// TIA Portal project "NodeRed_0" (V20)

(* hardware
DEVICE "S7-1500/ET200MP-Station_1"  S7-1500 station
   slot 0: "Profilschiene_0"  Rack  6ES7 590-1***0-0AA0
   slot 1: "PLC_1"  CPU 1515-2 PN  6ES7 515-2AM02-0AB0  V2.9
      slot 3: "CPU-Display_1"  6ES7591-1BA00-0AA0
      slot 32768: "PROFINET-Schnittstelle_1"  X1
         slot 32769: "Port_1"  X1 P1
         slot 32770: "Port_2"  X1 P2
      slot 33024: "PROFINET-Schnittstelle_2"  X2
         slot 33025: "Port_1"  X2 P1
      slot 34817: "Virtual CP interface port_1"  Virtual CP interface port  Virtual CP interface port
DEVICE "HMI_1"  TP700 Comfort
   slot 0: "HMI_1"  TP700 Comfort  6AV2 124-0GC01-0AX0  17.0.0.0
   slot 1: "HMI_RT_1"  TP700 Comfort  6AV2 124-0GC01-0AX0  17.0.0.0
   slot 5: "HMI_1.IE_CP_1"  PROFINET Interface  17.0.0.0
      slot 1: "PROFINET Schnittstelle_1"  PROFINET Interface
         slot 1: "Port_1"  Port
         slot 2: "Port_2"  Port
   slot 7: "HMI_1.MPI/DP_CP_1"  MPI/DP Interface  17.0.0.0
*)

// ===== PLC "PLC_1"  CPU 1515-2 PN =====

VAR_GLOBAL   // PLC tag table "Eingaenge"
   "2B1" AT %ED30 : DInt;   // Visionsensor
   "1B1" AT %E0.0 : Bool;   // Sensor_ein
   "3B1" AT %E0.1 : Bool;   // Sensor_aus
   "Factory/IO Running" AT %E0.7 : Bool;
END_VAR

VAR_GLOBAL   // PLC tag table "Ausgaenge"
   "1M1" AT %A0.0 : Bool;   // Band_1 (2m)
   "2M1" AT %A0.1 : Bool;   // Band_2 (2m)
   "3M1" AT %A0.2 : Bool;   // Band_3 (2m)
   "D1" AT %AD30 : DInt;   // Display
   "1H1" AT %A0.6 : Bool;   // Meldeleuchte (rot)
   "1H3" AT %A0.7 : Bool;   // Meldeleuchte (grün)
END_VAR

TYPE "typEingaenge"
   STRUCT
      "1B1" : Bool;
      "2B1" : DInt;
      "3B1" : Bool;
   END_STRUCT;
END_TYPE

TYPE "typAusgaenge"
   STRUCT
      "1M1" : Bool;
      "2M1" : Bool;
      "3M1" : Bool;
   END_STRUCT;
END_TYPE

TYPE "typZaehler"
   STRUCT
      Gesamt : DInt;
      Blau : Struct
         Gesamt : DInt;
         Roh : DInt;
         Oberteil : DInt;
         Unterteil : DInt;
      END_STRUCT;
      Gruen : Struct
         Gesamt : DInt;
         Roh : DInt;
         Oberteil : DInt;
         Unterteil : DInt;
      END_STRUCT;
      Metall : Struct
         Gesamt : DInt;
         Roh : DInt;
         Oberteil : DInt;
         Unterteil : DInt;
      END_STRUCT;
   END_STRUCT;
END_TYPE

DATA_BLOCK "IDB_Anlage_ein"   // DB1
{ S7_Optimized_Access := 'TRUE' }
VERSION : 0.1
// stored: InstanceOfName Anlage_ein
"Anlage_ein"
BEGIN
END_DATA_BLOCK

DATA_BLOCK "IDB_Bandsteuerung"   // DB10
{ S7_Optimized_Access := 'TRUE' }
VERSION : 0.1
// stored: InstanceOfName Bandsteuerung
"Bandsteuerung"
BEGIN
END_DATA_BLOCK

DATA_BLOCK "IDB_Bauteile_zaehlen"   // DB20
{ S7_Optimized_Access := 'TRUE' }
VERSION : 0.1
// stored: InstanceOfName Bauteile_zaehlen
"Bauteile_zaehlen"
BEGIN
END_DATA_BLOCK

DATA_BLOCK "HMI"   // DB100
{ S7_Optimized_Access := 'TRUE' }
VERSION : 0.1
   VAR
      Eingaenge : "typEingaenge";
      Ausgaenge : "typAusgaenge";
      Anlagedaten : Struct
         Anlage_aktiv : Bool;
         Laufzeit : DTL;
         Bauteile : "typZaehler";
         Bauteil : DInt;
      END_STRUCT;
   END_VAR
BEGIN
END_DATA_BLOCK

FUNCTION_BLOCK "Anlage_ein"   // FB1, FBD
{ S7_Optimized_Access := 'TRUE' }
VERSION : 0.1
BEGIN

REGION Network 1 (SCL)
   "HMI".Eingaenge."1B1" := "1B1";
   "HMI".Eingaenge."2B1" := "2B1";
   "HMI".Eingaenge."3B1" := "3B1";
END_REGION
END_FUNCTION_BLOCK

FUNCTION_BLOCK "Bandsteuerung"   // FB10, FBD
{ S7_Optimized_Access := 'TRUE' }
VERSION : 0.1
   VAR
      MI_RTRIG_FactoryRun : R_TRIG;
      MI_FTRIG_1B1 : F_TRIG;
      MI_FTRIG_3B1 : F_TRIG;
   END_VAR
BEGIN

REGION Network 1 (SCL): Flanken
   #MI_RTRIG_FactoryRun(CLK:="Factory/IO Running");

   #MI_FTRIG_1B1(CLK:="HMI".Eingaenge."1B1");
   #MI_FTRIG_3B1(CLK := "HMI".Eingaenge."3B1");
END_REGION

REGION Network 2 (SCL)
   "HMI".Ausgaenge."1M1" :=
   "HMI".Ausgaenge."2M1" :=
   "HMI".Ausgaenge."3M1" := #MI_RTRIG_FactoryRun.Q;
END_REGION
END_FUNCTION_BLOCK

FUNCTION_BLOCK "Bauteile_zaehlen"   // FB20, FBD
{ S7_Optimized_Access := 'TRUE' }
VERSION : 0.1
   VAR_INPUT
      Trigger : Bool;
      Bauteil : DInt;
   END_VAR
   VAR_IN_OUT
      Anzahl : "typZaehler";
   END_VAR
BEGIN

REGION Network 1 (SCL)
   IF #Trigger THEN
       CASE #Bauteil OF
           // Blaue Teile
           1:
               #Anzahl.Blau.Roh += 1;
           2:
               #Anzahl.Blau.Oberteil += 1;
           3:
               #Anzahl.Blau.Unterteil += 1;

           // Grüne Teile
           4:
               #Anzahl.Gruen.Roh += 1;
           5:
               #Anzahl.Gruen.Oberteil += 1;
           6:
               #Anzahl.Gruen.Unterteil += 1;

           // Metall Teile
           4:
               #Anzahl.Metall.Roh += 1;
           5:
               #Anzahl.Metall.Oberteil += 1;
           6:
               #Anzahl.Metall.Unterteil += 1;
       END_CASE;


       // Gesamtnanzahl einzelne Teile
       #Anzahl.Blau.Gesamt := #Anzahl.Blau.Roh
                           + #Anzahl.Blau.Oberteil
                           + #Anzahl.Blau.Unterteil;

       #Anzahl.Gruen.Gesamt := #Anzahl.Gruen.Roh
                           + #Anzahl.Gruen.Oberteil
                           + #Anzahl.Gruen.Unterteil;

       #Anzahl.Metall.Gesamt := #Anzahl.Metall.Roh
                           + #Anzahl.Metall.Oberteil
                           + #Anzahl.Metall.Unterteil;


       // Gesamtnanzahl alle Teile
       #Anzahl.Gesamt := #Anzahl.Metall.Gesamt
                       + #Anzahl.Gruen.Gesamt
                       + #Anzahl.Metall.Gesamt;
   END_IF;
END_REGION
END_FUNCTION_BLOCK

FUNCTION "Anlage_aus" : Void   // FC1, FBD
{ S7_Optimized_Access := 'TRUE' }
VERSION : 0.1
BEGIN

REGION Network 1 (SCL)
   // Bits
   "1M1" := "HMI".Ausgaenge."1M1";
   "2M1" := "HMI".Ausgaenge."2M1";
   "3M1" := "HMI".Ausgaenge."3M1";

   "Tag_1" := NOT "HMI".Anlagedaten.Anlage_aktiv;
   "Tag_2" := "HMI".Anlagedaten.Anlage_aktiv;


   // Word
   "D1" := "HMI".Anlagedaten.Anzahl_Bauteile.Gesamt;
END_REGION
END_FUNCTION

ORGANIZATION_BLOCK "Main"   // OB1, FBD, ProgramCycle
TITLE = "Main Program Sweep (Cycle)"
{ S7_Optimized_Access := 'TRUE' }
VERSION : 0.1
   VAR_INPUT
      Initial_Call : Bool;   // Initial call of this OB
      Remanence : Bool;   // =True, if remanent data are available
   END_VAR
BEGIN

REGION Network 1
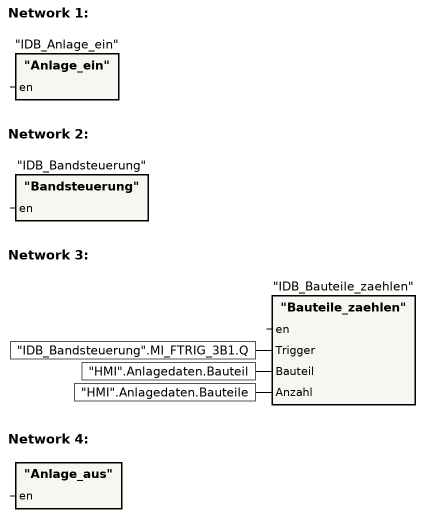
   "IDB_Anlage_ein"();   // "Anlage_ein"
END_REGION

REGION Network 2
   "IDB_Bandsteuerung"();   // "Bandsteuerung"
END_REGION

REGION Network 3
   "IDB_Bauteile_zaehlen"(Trigger := "IDB_Bandsteuerung".MI_FTRIG_3B1.Q,   // "Bauteile_zaehlen"
                          Bauteil := "HMI".Anlagedaten.Bauteil,
                          Anzahl := "HMI".Anlagedaten.Bauteile);
END_REGION

REGION Network 4
   "Anlage_aus"();
END_REGION
END_ORGANIZATION_BLOCK

(* ===== HMI "HMI_RT_1" =====
system functions are stored by id; their names below are inferred from use

HMI tags "Standard-Variablentabelle"
   "Variable_Bildnummer" : UInt, internal

text list "Textliste_Bildnamen": 1 'Home'; 2 'Anlagedaten'

screen "01_Home" 800x420, template "Menueleiste"
   on GenerateScreen: SetTag("Variable_Bildnummer", 1)

Template "Menueleiste" 800x420
   Button "Beenden" at 720,360 size 78x58; TextOff 'Beenden'; PictureOff "ExitRuntime_TP700_Comfort_TR"; PictureOn "ExitRuntime_TP700_Comfort_TR"
      on Release: StopRuntime(0)
   Button "Template_Button" at 640,360 size 78x58; TextOff 'Text'
   Button "Template_Button_1" at 560,360 size 78x58; TextOff 'Text'
   Button "Template_Button_2" at 480,360 size 78x58; TextOff 'Text'
   Button "Template_Button_3" at 400,360 size 78x58; TextOff 'Text'
   Button "Template_Button_4" at 321,360 size 78x58; TextOff 'Text'
   Button "Template_Button_5" at 241,360 size 78x58; TextOff 'Text'
   Button "Template_Button_6" at 161,360 size 78x58; TextOff 'Text'
   Button "Anlagedaten" at 81,360 size 78x58; TextOff 'Anlage'; PictureOff "Grafik_3"
      on Release: ActivateScreen("02_Anlagedaten", 0)
      on Press: SetTag("Variable_Bildnummer", 2)
      Appearance <- "Variable_Bildnummer"
   Button "Startbild" at 1,360 size 78x58; TextOff 'Startbild'; PictureOff "NavigateHome_TP700_Comfort_TR"; PictureOn "NavigateHome_TP700_Comfort_TR"
      on Release: ActivateScreen("01_Home", 0)
      on Press: SetTag("Variable_Bildnummer", 1)
      Appearance <- "Variable_Bildnummer"
*)